PROGRAM MAIN
VAR
	call : PLCOpenCall;
	command : PLCOpenCommand;
END_VAR

END_PROGRAM

(* stored: Version 1.1.0.1, ProductVersion 3.1.4024.12
   POU MAIN: Id {da7b43c9-38b1-4c6f-a60e-db64ccc086f5}, SpecialFunc None *)
